/// Project specific global var's
//{attribute 'qualified_only'}
VAR_GLOBAL
	// ToDo: comissioning
	iIBN : INT := 1;
	bTest : BOOL;
END_VAR

(* stored: Version 1.1.0.1
   GVL GVL: Id {f8176bf4-c77d-430d-b42e-51ee16e1ac45} *)
